(* PLC project OOP_Curso, Beckhoff Automation GmbH TwinCAT PLC Control 3.5.13.21 *)
(* stored: creationDateTime 2023-02-25T12:54:01.5537044, modificationDateTime 2023-02-25T12:54:01.5537044 *)

TYPE ST_sample2 :
STRUCT
	bbool	: BOOL;
	bVar 	: BOOL;
    nVar 	: INT;
	rreal 	: REAL;
	sstring : STRING;
END_STRUCT
END_TYPE

INTERFACE interface3
METHOD itf_metodo : BOOL
VAR_INPUT
END_VAR
END_METHOD
PROPERTY itf_propiedad : real
END_PROPERTY
END_INTERFACE

PROGRAM _05_Metodo
VAR
	fbejemplo_metodo : FB_ejemplo_Method;
	
	bPonerAUnobBoolfb : BOOL;
	bPonerACerobBoolfb: BOOL;
	
	bBool : BOOL;
	statusbBool : BOOL;
	bPonerAUnobBool : BOOL;
	bPonerACerobBool: BOOL;
	
	nSingleGet  : INT;
    stGet       : ST_Sample2;    
    bSet        : BOOL;
    stSet       : ST_Sample2;
	
	counter : INT;
	outvarcounter: INT;
END_VAR

            
IF 	bPonerAUnobBoolfb THEN
	bPonerAUnobBoolfb := FALSE;
	fbejemplo_metodo.metodo1_a_Uno_bBool();	
END_IF


IF 	bPonerACerobBoolfb THEN
	bPonerACerobBoolfb := FALSE;
	fbejemplo_metodo.metodo1_a_cero_bBool();
END_IF


IF 	bPonerAUnobBool THEN
	bPonerAUnobBool := FALSE;
	statusbBool := fbejemplo_metodo.metodo1_a_Uno_InOut(bBool);
END_IF

IF 	bPonerACerobBool THEN
	bPonerACerobBool := FALSE;
	statusbBool := fbejemplo_metodo.metodo1_a_Cero_InOut(bBool);
END_IF

// ejemplo para declarar variables lo mas cerca posible del metodo: declaración dentro del metodo de variable con VAR_INST :
counter := fbejemplo_metodo.Metodo4_VarInst(outvarcounter=>outvarcounter);

// Set and Get
IF bSet THEN  
	nSingleGet := fbejemplo_metodo.metodo2_struct(stSet).nVar;
	stGet      := fbejemplo_metodo.metodo2_struct(stSet);
	bSet            := FALSE;
END_IF  
          
END_PROGRAM

FUNCTION_BLOCK FB_ejemplo_Method
VAR_INPUT
END_VAR
VAR_OUTPUT
END_VAR
VAR
	bBool : BOOL;
	ststruct : ST_sample2;
	fb5 : fbreturn5;
END_VAR

            
          

METHOD metodo1_a_Cero_bBool
                  THIS^.bBool := false;
                
END_METHOD

METHOD metodo1_a_Cero_InOut : bool
VAR_IN_OUT
	bBool : BOOL;
END_VAR
                  // Método que pone a 0 la variable definida en in_Out
bBool := FALSE;
// return value bBOOL
metodo1_a_Cero_InOut := FALSE;
                
END_METHOD

METHOD metodo1_a_Uno_bBool
                  THIS^.bBool := true;
                
END_METHOD

METHOD metodo1_a_Uno_InOut : BOOL
VAR_IN_OUT
	bBool : BOOL;
END_VAR
                  // Método que pone a 1 la variable definida en in_Out
bBool := TRUE;
// return value bBOOL
metodo1_a_Uno_InOut := TRUE;
                
END_METHOD

METHOD PUBLIC metodo2_struct : REFERENCE TO ST_sample2
VAR_INPUT
	st_struct : ST_sample2;
END_VAR
                  

THIS^.ststruct := st_struct;

metodo2_struct REF= THIS^.ststruct;
                
END_METHOD

METHOD PRIVATE metodo3_interface : interface3
VAR_INPUT
END_VAR
                  


                
END_METHOD

METHOD Metodo4_VarInst : INT
VAR_OUTPUT
	outvarcounter : INT;
END_VAR
VAR
	varcounter : INT;
END_VAR
VAR_INST
	counter : INT;
END_VAR
                  counter := counter + 1;
Metodo4_VarInst := counter;

varcounter := varcounter + 1; 
outvarcounter := varcounter; 


                
END_METHOD

METHOD metodo5_returnfb : fbreturn5
VAR_INPUT
END_VAR
                  metodo5_returnfb := fb5;
                
END_METHOD

METHOD metodo0_Declaracion_variables
VAR_INPUT
	binput : BOOL;
END_VAR
VAR_INPUT
	binput2 : BOOL;
END_VAR
VAR_OUTPUT
	output1 : REAL;
END_VAR
VAR_IN_OUT
	in_out1 : LINT;
END_VAR
VAR_IN_OUT CONSTANT
	in_out_constant1 : DINT;
END_VAR
VAR
	var1 : STRING;
END_VAR
//!!! no se pueden declarar variables TEMPORALES dentro de la zona de declaración de variables del método!!!
//VAR_TEMP
//	temp1 : ULINT;
//END_VAR
VAR_INST
	counter : INT;
END_VAR
VAR_STAT
    nVarStat1 : INT;
	aarray  : ARRAY[1..n] OF INT;
END_VAR
VAR_EXTERNAL
    nVarExt1 : INT; // 1st external variable
END_VAR
//!!! no se pueden declarar variables PERSISTENT ni RETAIN dentro de la zona de declaración de variables del método!!!
//VAR PERSISTENT
//    nVarPers1 : DINT; (* 1. Persistent variable *)
//    bVarPers2 : BOOL; (* 2. Persistent variable *)
//END_VAR
//VAR RETAIN
//    nRem1 : INT;
//END_VAR
VAR CONSTANT
	n : INT:= 10;
END_VAR
                  
                
END_METHOD
END_FUNCTION_BLOCK

FUNCTION_BLOCK fbreturn5
VAR_INPUT
END_VAR
VAR_OUTPUT
END_VAR
VAR
END_VAR

            
          
END_FUNCTION_BLOCK
